TYPE TcaSingleAxisRef :
STRUCT
	tsAcknowledge AT%Q* : BOOL;
	tsAcknowledgeRequest AT%I* : BOOL;
	tsSS1Active AT%I* : BOOL;
	tsSTOActive AT%I* : BOOL;	
END_STRUCT
END_TYPE

(* stored: Version 1.1.0.1
   DUT TcaSingleAxisRef: Id {3c8b2ff9-9380-4582-aded-18a42867d38d} *)
